// TIA Portal V20 export
FUNCTION "Fx_LadInterlock" : Void   // FC10, LAD
{ S7_Optimized_Access := 'TRUE' }
   VAR_INPUT
      Enable : Bool;
      Guard : Bool;
   END_VAR
   VAR_OUTPUT
      Out : Bool;
   END_VAR
BEGIN

REGION Network 1
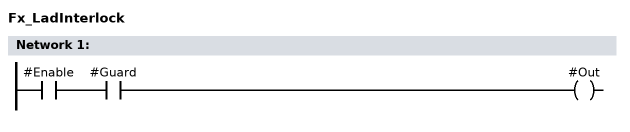
   RUNG wire#powerrail
      Contact( #Enable )
      Contact( #Guard )
      Coil( #Out )
   END_RUNG
   // the same network as SCL:
   #Out := #Enable AND #Guard;
END_REGION
END_FUNCTION
